(* CoDeSys 2.3.9.62 project: ControlNivelDosBombas v0.pro *)

(* Global variable list: Global_Variables *)
VAR_GLOBAL

(* Entradas *)
     A:BOOL;
     B:BOOL;
     Encendido:BOOL;

(*Salidas *)
  Bomba1:BOOL;
  Bomba2:BOOL;

END_VAR

(* POU PLC_PRG, ST *)
PROGRAM PLC_PRG
VAR

END_VAR
Control();
Simulacion();
END_PROGRAM

(* POU Control, LD *)
PROGRAM Control
VAR
	E0: BOOL;
	E1: BOOL;
	E2: BOOL;
	E3: BOOL;
	E4: BOOL;
	E5: BOOL;
	E6: BOOL;
	B1: BOOL;
	B2: BOOL;
	B3: BOOL;
END_VAR
VAR (* helpers for the ST form of the networks *)
	_p1 : BOOL;
	_p2 : BOOL;
	_p3 : BOOL;
	_p4 : BOOL;
	_p5 : BOOL;
	_p6 : BOOL;
	_p7 : BOOL;
END_VAR
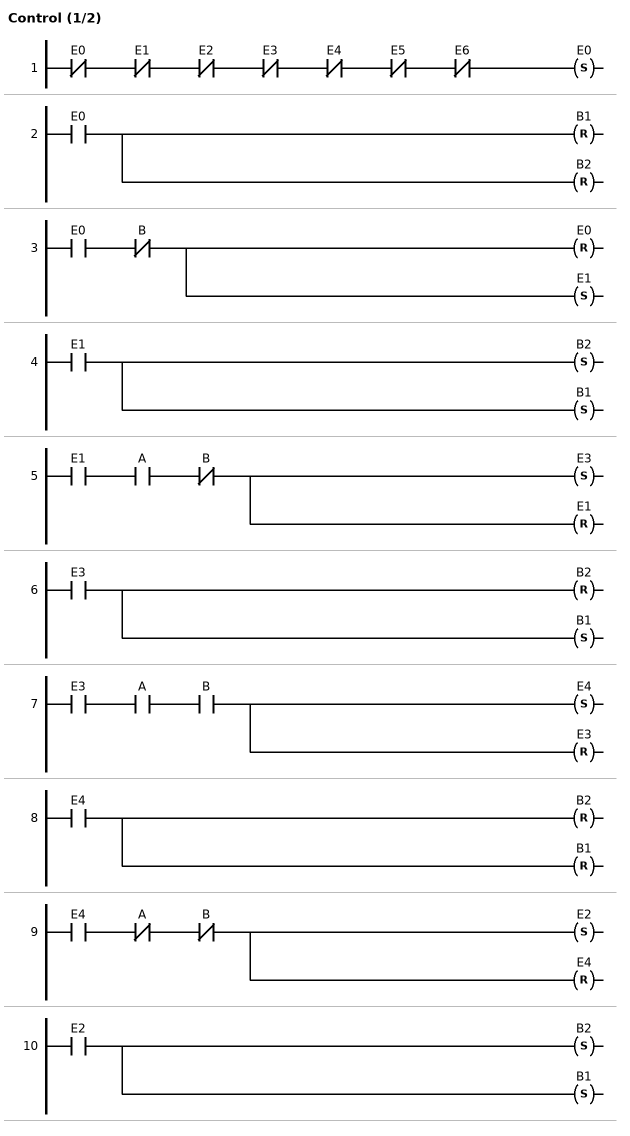
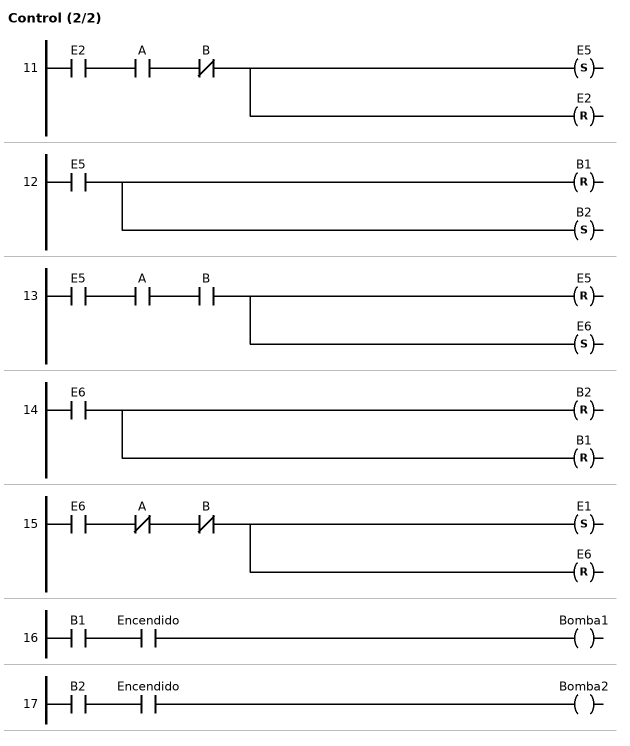
_LD_ (* Ladder Diagram *)
NETWORK 1
	[/E0] - [/E1] - [/E2] - [/E3] - [/E4] - [/E5] - [/E6] --- (S E0)
NETWORK 2
	[E0] --- (R B1) (R B2)
NETWORK 3
	[E0] - [/B] --- (R E0) (S E1)
NETWORK 4
	[E1] --- (S B2) (S B1)
NETWORK 5
	[E1] - [A] - [/B] --- (S E3) (R E1)
NETWORK 6
	[E3] --- (R B2) (S B1)
NETWORK 7
	[E3] - [A] - [B] --- (S E4) (R E3)
NETWORK 8
	[E4] --- (R B2) (R B1)
NETWORK 9
	[E4] - [/A] - [/B] --- (S E2) (R E4)
NETWORK 10
	[E2] --- (S B2) (S B1)
NETWORK 11
	[E2] - [A] - [/B] --- (S E5) (R E2)
NETWORK 12
	[E5] --- (R B1) (S B2)
NETWORK 13
	[E5] - [A] - [B] --- (R E5) (S E6)
NETWORK 14
	[E6] --- (R B2) (R B1)
NETWORK 15
	[E6] - [/A] - [/B] --- (S E1) (R E6)
NETWORK 16
	[B1] - [Encendido] --- (Bomba1)
NETWORK 17
	[B2] - [Encendido] --- (Bomba2)
_END_LD_
(* the same logic as Structured Text *)
(* Network 1 *)
IF NOT E0 AND NOT E1 AND NOT E2 AND NOT E3 AND NOT E4 AND NOT E5 AND NOT E6 THEN E0 := TRUE; END_IF;
(* Network 2 *)
IF E0 THEN B1 := FALSE; B2 := FALSE; END_IF;
(* Network 3 *)
_p1 := E0 AND NOT B;
IF _p1 THEN E0 := FALSE; E1 := TRUE; END_IF;
(* Network 4 *)
IF E1 THEN B2 := TRUE; B1 := TRUE; END_IF;
(* Network 5 *)
_p2 := E1 AND A AND NOT B;
IF _p2 THEN E3 := TRUE; E1 := FALSE; END_IF;
(* Network 6 *)
IF E3 THEN B2 := FALSE; B1 := TRUE; END_IF;
(* Network 7 *)
_p3 := E3 AND A AND B;
IF _p3 THEN E4 := TRUE; E3 := FALSE; END_IF;
(* Network 8 *)
IF E4 THEN B2 := FALSE; B1 := FALSE; END_IF;
(* Network 9 *)
_p4 := E4 AND NOT A AND NOT B;
IF _p4 THEN E2 := TRUE; E4 := FALSE; END_IF;
(* Network 10 *)
IF E2 THEN B2 := TRUE; B1 := TRUE; END_IF;
(* Network 11 *)
_p5 := E2 AND A AND NOT B;
IF _p5 THEN E5 := TRUE; E2 := FALSE; END_IF;
(* Network 12 *)
IF E5 THEN B1 := FALSE; B2 := TRUE; END_IF;
(* Network 13 *)
_p6 := E5 AND A AND B;
IF _p6 THEN E5 := FALSE; E6 := TRUE; END_IF;
(* Network 14 *)
IF E6 THEN B2 := FALSE; B1 := FALSE; END_IF;
(* Network 15 *)
_p7 := E6 AND NOT A AND NOT B;
IF _p7 THEN E1 := TRUE; E6 := FALSE; END_IF;
(* Network 16 *)
Bomba1 := B1 AND Encendido;
(* Network 17 *)
Bomba2 := B2 AND Encendido;
END_PROGRAM

(* POU Simulacion, ST *)
PROGRAM Simulacion
VAR
   posy:INT;
	PrimerCiclo: BOOL:=TRUE;
	posInicial: INT;
END_VAR
IF posy>-187 THEN
IF (Bomba1=TRUE AND Bomba2=TRUE) THEN
  posy:=posy-2;
ELSE
     IF (Bomba1=TRUE OR Bomba2=TRUE) THEN
            posy:=posy-1;
     END_IF
END_IF
END_IF

IF (Bomba1=FALSE AND Bomba2=FALSE) THEN
IF posy<52 THEN
  posy:=posy+1;
END_IF
END_IF



IF posy<-50 THEN
  A:=TRUE;
ELSE
  A:=FALSE;
END_IF

IF posy<=-164 THEN
  B:=TRUE;
ELSE
  B:=FALSE;
END_IF

(* Solo en primer ciclo*)
IF (PrimerCiclo) THEN
    PrimerCiclo:=FALSE;
    posy:=posInicial;
END_IF
END_PROGRAM

(* Visualisation Deposito
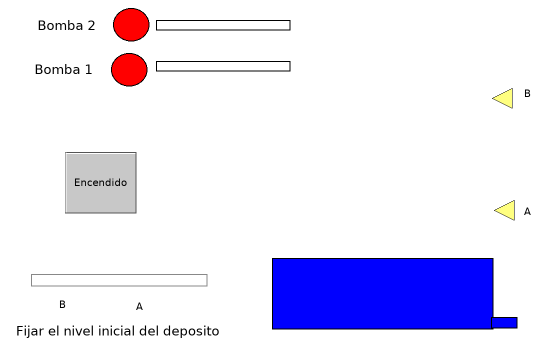
button at (94,178)-(165,239): text "Encendido"; toggles .Encendido
polygon at (521,114)-(541,134): alarm colour if .B; toggles .B
polygon at (523,226)-(543,246): alarm colour if .A; toggles .A
rectangle at (301,284)-(522,355): top Simulacion.posy
rectangle at (541,222)-(572,253): text "A"
rectangle at (541,104)-(572,135): text "B"
rectangle at (185,87)-(319,97): alarm colour if Bomba1
rectangle at (185,46)-(319,56): alarm colour if Bomba2
ellipse at (140,79)-(176,112): alarm colour if Bomba1
ellipse at (142,34)-(178,67): alarm colour if Bomba2
rectangle at (48,80)-(138,111): text "Bomba 1"
rectangle at (51,36)-(141,67): text "Bomba 2"
rectangle at (76,315)-(107,346): text "B"
rectangle at (153,317)-(184,348): text "A"
rectangle at (39,343)-(255,371): text "Fijar el nivel inicial del deposito"
4 more shapes without text or variables
*)
